LIN {X 0,Y 23.912,Z 617.409,A -85,B 0,C 180,E1 -30546.001,E2 -30546.001} C_VEL
LIN {X 0,Y 33.285,Z 615.742,A -85,B 0,C 180,E1 -30567.625,E2 -30567.625} C_VEL
LIN {X 0,Y 45.152,Z 612.913,A -85,B 0,C 180,E1 -30579.05,E2 -30579.05} C_VEL
LIN {X 0,Y 58.951,Z 608.498,A -85,B 0,C 180,E1 -30586.205,E2 -30586.205} C_VEL
LIN {X 0,Y 71.331,Z 603.47,A -85,B 0,C 180,E1 -30590.142,E2 -30590.142} C_VEL
LIN {X 0,Y 84.935,Z 596.599,A -85,B 0,C 180,E1 -30593.175,E2 -30593.175} C_VEL
LIN {X 0,Y 96.989,Z 589.21,A -85,B 0,C 180,E1 -30595.087,E2 -30595.087} C_VEL
LIN {X 0,Y 105.632,Z 582.993,A -85,B 0,C 180,E1 -30596.342,E2 -30596.342} C_VEL
LIN {X 0,Y 117.82,Z 572.82,A -85,B 0,C 180,E1 -30597.591,E2 -30597.591} C_VEL
LIN {X 0,Y 128.3,Z 562.41,A -85,B 0,C 180,E1 -30598.52,E2 -30598.52} C_VEL
LIN {X 0,Y 137.933,Z 551.077,A -85,B 0,C 180,E1 -30599.228,E2 -30599.228} C_VEL
LIN {X 0,Y 140.563,Z 547.571,A -85,B 0,C 180,E1 -30599.436,E2 -30599.436} C_VEL
LIN {X 0,Y 140.56,Z 547.579,A -85,B 0,C 180,E1 -30599.555,E2 -30599.555} C_VEL
LIN {X 0,Y 130.771,Z 559.725,A -85,B 0,C 180,E1 -30600.205,E2 -30600.205} C_VEL
LIN {X 0,Y 121.244,Z 569.76,A -85,B 0,C 180,E1 -30600.897,E2 -30600.897} C_VEL
LIN {X 0,Y 110.739,Z 579.149,A -85,B 0,C 180,E1 -30601.735,E2 -30601.735} C_VEL
LIN {X 0,Y 98.527,Z 588.389,A -85,B 0,C 180,E1 -30603.031,E2 -30603.031} C_VEL
LIN {X 0,Y 87.168,Z 595.622,A -85,B 0,C 180,E1 -30604.624,E2 -30604.624} C_VEL
LIN {X 0,Y 74.377,Z 602.471,A -85,B 0,C 180,E1 -30607.191,E2 -30607.191} C_VEL
LIN {X 0,Y 60.831,Z 608.347,A -85,B 0,C 180,E1 -30610.884,E2 -30610.884} C_VEL
LIN {X 0,Y 50.931,Z 611.852,A -85,B 0,C 180,E1 -30615.002,E2 -30615.002} C_VEL
LIN {X 0,Y 38.363,Z 615.401,A -85,B 0,C 180,E1 -30623.658,E2 -30623.658} C_VEL
LIN {X 0,Y 27.354,Z 617.746,A -85,B 0,C 180,E1 -30639.579,E2 -30639.579} C_VEL
LIN {X 0,Y 20.524,Z 618.943,A -85,B 0,C 180,E1 -30669.975,E2 -30669.975} C_VEL
LIN {X 0,Y 19.929,Z 619.111,A -85,B 0,C 180,E1 -30690,E2 -30690} C_VEL
LIN {X 0,Y 23.146,Z 618.462,A -85,B 0,C 180,E1 -30727.392,E2 -30727.392} C_VEL
LIN {X 0,Y 32.548,Z 616.663,A -85,B 0,C 180,E1 -30749.733,E2 -30749.733} C_VEL
LIN {X 0,Y 45.536,Z 613.399,A -85,B 0,C 180,E1 -30762.021,E2 -30762.021} C_VEL
LIN {X 0,Y 57.504,Z 609.495,A -85,B 0,C 180,E1 -30767.88,E2 -30767.88} C_VEL
LIN {X 0,Y 70.968,Z 603.949,A -85,B 0,C 180,E1 -30772.002,E2 -30772.002} C_VEL
LIN {X 0,Y 84.673,Z 596.907,A -85,B 0,C 180,E1 -30774.869,E2 -30774.869} C_VEL
LIN {X 0,Y 96.787,Z 589.383,A -85,B 0,C 180,E1 -30776.761,E2 -30776.761} C_VEL
LIN {X 0,Y 108.993,Z 580.328,A -85,B 0,C 180,E1 -30778.066,E2 -30778.066} C_VEL
LIN {X 0,Y 119.491,Z 571.085,A -85,B 0,C 180,E1 -30778.999,E2 -30778.999} C_VEL
LIN {X 0,Y 129.47,Z 560.809,A -85,B 0,C 180,E1 -30779.722,E2 -30779.722} C_VEL
LIN {X 0,Y 139.681,Z 548.319,A -85,B 0,C 180,E1 -30780.397,E2 -30780.397} C_VEL
LIN {X 0,Y 140.56,Z 547.142,A -85,B 0,C 180,E1 -30780.449,E2 -30780.449} C_VEL
LIN {X 0,Y 140.565,Z 547.129,A -85,B 0,C 180,E1 -30780.639,E2 -30780.639} C_VEL
LIN {X 0,Y 140.603,Z 549.128,A -85,B 0,C 180,E1 -30781.477,E2 -30781.477} C_VEL
LIN {X 0,Y 140.603,Z 602.402,A -85,B 0,C 180,E1 -30781.477,E2 -30781.477} C_VEL
LIN {X 0,Y 96.405,Z 602.402,A -85,B 0,C 180,E1 -30781.136,E2 -30781.136} C_VEL
LIN {X 0,Y 94.405,Z 600.402,A -85,B 0,C 180,E1 -30781.113,E2 -30781.113} C_VEL
LIN {X 0,Y 94.405,Z 594.219,A -85,B 0,C 180,E1 -30781.113,E2 -30781.113} C_VEL
LIN {X 0,Y 91.387,Z 592.514,A -85,B 0,C 180,E1 -30781.366,E2 -30781.366} C_VEL
LIN {X 0,Y 80.901,Z 598.461,A -85,B 0,C 180,E1 -30782.575,E2 -30782.575} C_VEL
LIN {X 0,Y 67.003,Z 604.997,A -85,B 0,C 180,E1 -30784.837,E2 -30784.837} C_VEL
LIN {X 0,Y 53.263,Z 610.094,A -85,B 0,C 180,E1 -30788.274,E2 -30788.274} C_VEL
LIN {X 0,Y 43.127,Z 613.027,A -85,B 0,C 180,E1 -30792.116,E2 -30792.116} C_VEL
LIN {X 0,Y 30.102,Z 615.884,A -85,B 0,C 180,E1 -30800.953,E2 -30800.953} C_VEL
LIN {X 0,Y 18.647,Z 617.585,A -85,B 0,C 180,E1 -30821.084,E2 -30821.084} C_VEL
LIN {X 0,Y 13.054,Z 618.168,A -85,B 0,C 180,E1 -30870,E2 -30870} C_VEL
LIN {X 0,Y 18.641,Z 617.611,A -85,B 0,C 180,E1 -30918.94,E2 -30918.94} C_VEL
LIN {X 0,Y 30.071,Z 615.946,A -85,B 0,C 180,E1 -30939.199,E2 -30939.199} C_VEL
LIN {X 0,Y 43.12,Z 613.116,A -85,B 0,C 180,E1 -30947.929,E2 -30947.929} C_VEL
LIN {X 0,Y 57.012,Z 608.936,A -85,B 0,C 180,E1 -30952.918,E2 -30952.918} C_VEL
LIN {X 0,Y 70.462,Z 603.672,A -85,B 0,C 180,E1 -30955.858,E2 -30955.858} C_VEL
LIN {X 0,Y 84.386,Z 596.802,A -85,B 0,C 180,E1 -30957.988,E2 -30957.988} C_VEL
LIN {X 0,Y 91.386,Z 592.735,A -85,B 0,C 180,E1 -30958.682,E2 -30958.682} C_VEL
LIN {X 0,Y 91.366,Z 592.77,A -85,B 0,C 180,E1 -30959.455,E2 -30959.455} C_VEL
LIN {X 0,Y 77.321,Z 600.593,A -85,B 0,C 180,E1 -30961.135,E2 -30961.135} C_VEL
LIN {X 0,Y 63.361,Z 606.82,A -85,B 0,C 180,E1 -30963.384,E2 -30963.384} C_VEL
LIN {X 0,Y 49.559,Z 611.648,A -85,B 0,C 180,E1 -30966.949,E2 -30966.949} C_VEL
LIN {X 0,Y 36.089,Z 615.196,A -85,B 0,C 180,E1 -30973.177,E2 -30973.177} C_VEL
LIN {X 0,Y 23.448,Z 617.542,A -85,B 0,C 180,E1 -30985.952,E2 -30985.952} C_VEL
LIN {X 0,Y 14.025,Z 618.739,A -85,B 0,C 180,E1 -31019.928,E2 -31019.928} C_VEL
LIN {X 0,Y 12.818,Z 618.907,A -85,B 0,C 180,E1 -31050,E2 -31050} C_VEL
LIN {X 0,Y 17.997,Z 618.258,A -85,B 0,C 180,E1 -31101.35,E2 -31101.35} C_VEL
LIN {X 0,Y 29.592,Z 616.458,A -85,B 0,C 180,E1 -31121.796,E2 -31121.796} C_VEL
LIN {X 0,Y 42.923,Z 613.443,A -85,B 0,C 180,E1 -31130.577,E2 -31130.577} C_VEL
LIN {X 0,Y 56.437,Z 609.289,A -85,B 0,C 180,E1 -31135.005,E2 -31135.005} C_VEL
LIN {X 0,Y 70.331,Z 603.744,A -85,B 0,C 180,E1 -31137.78,E2 -31137.78} C_VEL
LIN {X 0,Y 84.334,Z 596.7,A -85,B 0,C 180,E1 -31139.74,E2 -31139.74} C_VEL
LIN {X 0,Y 91.365,Z 592.552,A -85,B 0,C 180,E1 -31140.545,E2 -31140.545} C_VEL
LIN {X 0,Y 91.387,Z 592.514,A -85,B 0,C 180,E1 -31141.366,E2 -31141.366} C_VEL
LIN {X 0,Y 91.459,Z 594.513,A -85,B 0,C 180,E1 -31142.655,E2 -31142.655} C_VEL
LIN {X 0,Y 91.459,Z 621.365,A -85,B 0,C 180,E1 -31142.655,E2 -31142.655} C_VEL
LIN {X 0,Y 52.666,Z 621.365,A -85,B 0,C 180,E1 -31140.893,E2 -31140.893} C_VEL
LIN {X 0,Y 50.672,Z 619.365,A -85,B 0,C 180,E1 -31140.73,E2 -31140.73} C_VEL
LIN {X 0,Y 50.672,Z 613.587,A -85,B 0,C 180,E1 -31140.73,E2 -31140.73} C_VEL
LIN {X 0,Y 48.204,Z 611.651,A -85,B 0,C 180,E1 -31141.211,E2 -31141.211} C_VEL
LIN {X 0,Y 35.247,Z 614.809,A -85,B 0,C 180,E1 -31144.485,E2 -31144.485} C_VEL
LIN {X 0,Y 21.545,Z 617.08,A -85,B 0,C 180,E1 -31151.887,E2 -31151.887} C_VEL
LIN {X 0,Y 9.028,Z 618.222,A -85,B 0,C 180,E1 -31178.879,E2 -31178.879} C_VEL
LIN {X 0,Y 5.959,Z 618.371,A -85,B 0,C 180,E1 -31230.001,E2 -31230.001} C_VEL
LIN {X 0,Y 14.958,Z 617.815,A -85,B 0,C 180,E1 -31299.996,E2 -31299.996} C_VEL
LIN {X 0,Y 28.333,Z 616.15,A -85,B 0,C 180,E1 -31312.829,E2 -31312.829} C_VEL
LIN {X 0,Y 42.209,Z 613.319,A -85,B 0,C 180,E1 -31317.428,E2 -31317.428} C_VEL
LIN {X 0,Y 47.965,Z 611.825,A -85,B 0,C 180,E1 -31318.844,E2 -31318.844} C_VEL
LIN {X 0,Y 35.155,Z 614.992,A -85,B 0,C 180,E1 -31321.734,E2 -31321.734} C_VEL
LIN {X 0,Y 21.31,Z 617.337,A -85,B 0,C 180,E1 -31328.366,E2 -31328.366} C_VEL
LIN {X 0,Y 8.627,Z 618.535,A -85,B 0,C 180,E1 -31355.451,E2 -31355.451} C_VEL
LIN {X 0,Y 5.697,Z 618.704,A -85,B 0,C 180,E1 -31409.999,E2 -31409.999} C_VEL
LIN {X 0,Y 14.635,Z 618.053,A -85,B 0,C 180,E1 -31483.819,E2 -31483.819} C_VEL
LIN {X 0,Y 28.187,Z 616.252,A -85,B 0,C 180,E1 -31495.783,E2 -31495.783} C_VEL
LIN {X 0,Y 42.167,Z 613.284,A -85,B 0,C 180,E1 -31500.149,E2 -31500.149} C_VEL
LIN {X 0,Y 48.204,Z 611.651,A -85,B 0,C 180,E1 -31501.211,E2 -31501.211} C_VEL
LIN {X 0,Y 48.204,Z 611.651,A -85,B 0,C 180,E1 -31501.211,E2 -31501.211}

QRS_NEXT_CUT()

QRS_NEXT()
QRS_HOME()

END
